FUNCTION_BLOCK TcLogTRIG EXTENDS TcLog
VAR_INPUT
END_VAR
VAR_OUTPUT
END_VAR
VAR
END_VAR

// Logs data on falling edge of CLK.
METHOD OnFallingEdge : REFERENCE TO TcLog
VAR_INPUT
	CLK 	:	BOOL;	// Falling edge logs data.
END_VAR
VAR_INST
	fTrig	:	F_TRIG;
END_VAR
fTrig(CLK:=CLK);

SUPER^.OnCondition(fTrig.Q);

OnFallingEdge REF= THIS^;
END_METHOD

// Logs data on rising edge of CLK.
METHOD OnRisingEdge : REFERENCE TO TcLog
VAR_INPUT
	CLK 	:	BOOL;		// Rising edge logs data.
END_VAR
VAR_INST
	rTrig	:	R_TRIG;
END_VAR
rTrig(CLK:=CLK);

SUPER^.OnCondition(rTrig.Q);

OnRisingEdge REF= THIS^;
END_METHOD

END_FUNCTION_BLOCK

(* stored: Version 1.1.0.1, ProductVersion 3.1.4024.4
   POU TcLogTRIG: Id {aef804a0-ffc6-4577-b368-1ac5b4e5d860}, SpecialFunc None
   Method OnFallingEdge: Id {a776a649-e65d-434f-b5b2-64de81890120}
   Method OnRisingEdge: Id {e0a21764-11de-45ad-894f-c14b1933c3ef} *)
